// TIA Portal project "lab6.8" (V15)

(* hardware
DEVICE "S7-1200 station_1"  S7-1200 Station
   slot 0: "Rack_0"  S7-1200 Rack  Rack  V1.0
   slot 1: "PLC_1"  CPU 1214C DC/DC/DC  6ES7 214-1AG40-0XB0  V4.2
      slot 3: "AQ 1x12BIT_1"  AQ1 signal board  6ES7 232-4HA30-0XB0  V1.0
   slot 101: "CM 1243-5"  CM 1243-5  6GK7 243-5DX30-0XE0  V1.3
   slot 102: "CM 1241 (RS485)_1"  CM 1241 (RS485)  6ES7 241-1CH30-0XB0  V1.0
*)

// ===== PLC "PLC_1"  CPU 1214C DC/DC/DC =====

VAR_GLOBAL   // PLC tag table "Default tag table"
   "startStop" AT %I0.1 : Bool;
   "zbocze" AT %M10.0 : Bool;
   "podzielnik" AT %M10.1 : Bool;
   "zwrot" AT %M10.2 : Bool;
   "sprzezenie" AT %M10.3 : Bool;
   "Tag_1" AT %Q0.6 : Bool;
   "Tag_2" AT %Q0.7 : Bool;
   "licznik" AT %M10.6 : Bool;
   "reset" AT %M10.5 : Bool;
END_VAR

// folder: System blocks/Program resources

DATA_BLOCK "t1"   // DB1
{ S7_Optimized_Access := 'TRUE' }
AUTHOR : Simatic
FAMILY : IEC
NAME : IEC_TMR
VERSION : 1.0
// stored: InstanceOfName IEC_TIMER
"IEC_TIMER"
BEGIN
END_DATA_BLOCK

DATA_BLOCK "t2"   // DB2
{ S7_Optimized_Access := 'TRUE' }
AUTHOR : Simatic
FAMILY : IEC
NAME : IEC_TMR
VERSION : 1.0
// stored: InstanceOfName IEC_TIMER
"IEC_TIMER"
BEGIN
END_DATA_BLOCK

DATA_BLOCK "C1"   // DB3
{ S7_Optimized_Access := 'TRUE' }
AUTHOR : Simatic
FAMILY : IEC
NAME : CNTR
VERSION : 1.0
// stored: InstanceOfName IEC_COUNTER
"IEC_COUNTER"
BEGIN
END_DATA_BLOCK

DATA_BLOCK "t3"   // DB4
{ S7_Optimized_Access := 'TRUE' }
AUTHOR : Simatic
FAMILY : IEC
NAME : IEC_TMR
VERSION : 1.0
// stored: InstanceOfName IEC_TIMER
"IEC_TIMER"
BEGIN
END_DATA_BLOCK

// folder: (top level)

ORGANIZATION_BLOCK "Main"   // OB1, LAD, ProgramCycle
TITLE = "Main Program Sweep (Cycle)"
{ S7_Optimized_Access := 'TRUE' }
VERSION : 0.1
// zbuduj generator wl i wyl jednym przyciskiem o f = 2Hz i wypelnieniu 20% (Q0.6) [p zliczeniu 15 impulsow automatycznie wylacz generator i sygnalizuj zliczenie przez czas 2s na wyjsciu Q0.7
   VAR_INPUT
      Initial_Call : Bool;   // Initial call of this OB
      Remanence : Bool;   // =True, if remanent data are available
   END_VAR
   VAR_TEMP   // added for the SCL form of the ladder/FBD networks
      _w1 : Bool;
   END_VAR
BEGIN

REGION Network 1: podzielnik binary
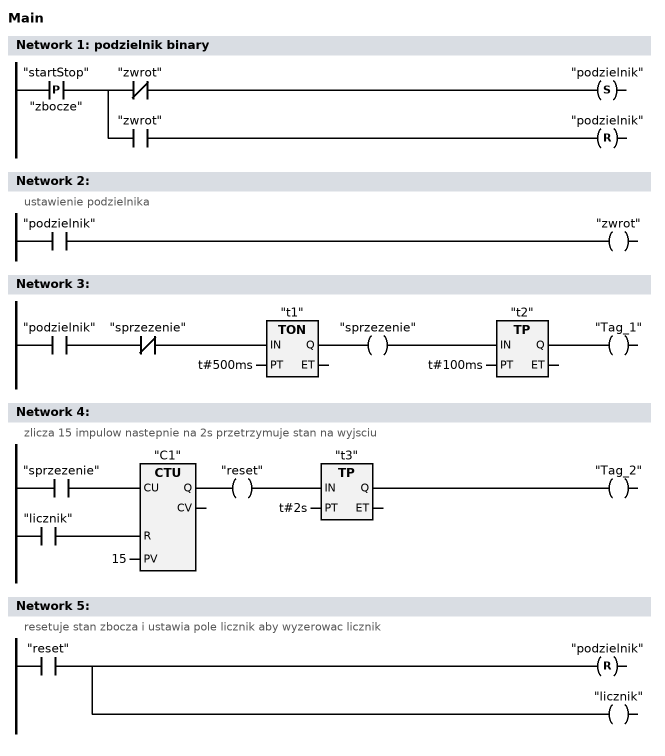
   RUNG wire#powerrail
      P_Contact(operand := "startStop", bit := "zbocze")
      wire#w1
      I_Contact( "zwrot" )
      S_Coil( "podzielnik" )
   END_RUNG
   RUNG wire#w1
      Contact( "zwrot" )
      R_Coil( "podzielnik" )
   END_RUNG
   // the same network as SCL:
   #_w1 := "startStop" AND NOT "zbocze";   // rising edge of "startStop"
   "zbocze" := "startStop";
   IF #_w1 AND NOT "zwrot" THEN "podzielnik" := TRUE; END_IF;
   IF #_w1 AND "zwrot" THEN "podzielnik" := FALSE; END_IF;
END_REGION

REGION Network 2
   // ustawienie podzielnika
   RUNG wire#powerrail
      Contact( "podzielnik" )
      Coil( "zwrot" )
   END_RUNG
   // the same network as SCL:
   "zwrot" := "podzielnik";
END_REGION

REGION Network 3
   "t1".TON(IN := "podzielnik" AND NOT "sprzezenie", PT := t#500ms);
   "sprzezenie" := "t1".Q;
   "t2".TP(IN := "t1".Q, PT := t#100ms);
   "Tag_1" := "t2".Q;
END_REGION

REGION Network 4
   // zlicza 15 impulow nastepnie na 2s przetrzymuje stan na wyjsciu
   "C1".CTU(CU := "sprzezenie", R := "licznik", PV := 15);
   "reset" := "C1".Q;
   "t3".TP(IN := "C1".Q, PT := t#2s);
   "Tag_2" := "t3".Q;
END_REGION

REGION Network 5
   // resetuje stan zbocza i ustawia pole licznik aby wyzerowac licznik
   RUNG wire#powerrail
      Contact( "reset" )
      wire#w1
      R_Coil( "podzielnik" )
   END_RUNG
   RUNG wire#w1
      Coil( "licznik" )
   END_RUNG
   // the same network as SCL:
   IF "reset" THEN "podzielnik" := FALSE; END_IF;
   "licznik" := "reset";
END_REGION
END_ORGANIZATION_BLOCK